FUNCTION_BLOCK CMP_OC_W4

VAR_INPUT
	BOOL_INTERLOCK : BOOL; (*INTERLOCK*)
	WORD_1: WORD;		(*WORD 1*)
	WORD_2: WORD;		(*WORD 2*)
	WORD_3: WORD;		(*WORD 3*)
	WORD_4: WORD;		(*WORD 4*)
	END_VAR


VAR_OUTPUT
	BZ_OUTPUT_BOOL : BOOL;
END_VAR


VAR
	OUT_1: BOOL;
	OUT_2: BOOL;
	OUT_3: BOOL;
	OUT_4: BOOL;
END_VAR

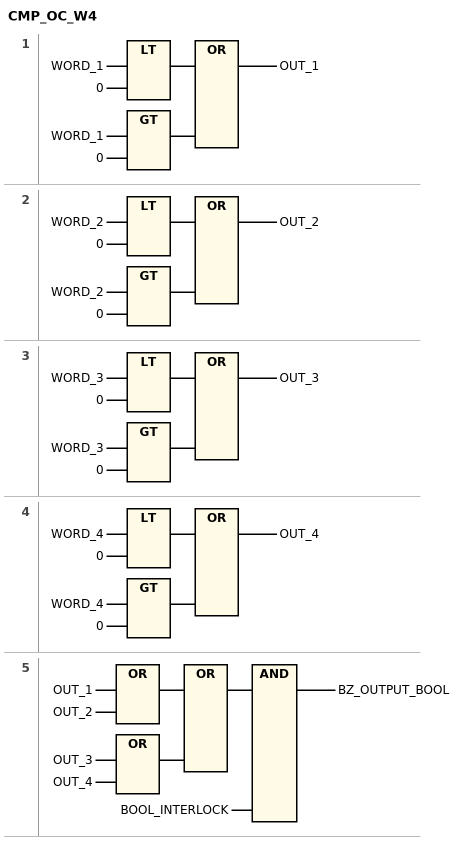
// NETWORK 1
OUT_1 := WORD_1 < 0 OR WORD_1 > 0;

// NETWORK 2
OUT_2 := WORD_2 < 0 OR WORD_2 > 0;

// NETWORK 3
OUT_3 := WORD_3 < 0 OR WORD_3 > 0;

// NETWORK 4
OUT_4 := WORD_4 < 0 OR WORD_4 > 0;

// NETWORK 5
BZ_OUTPUT_BOOL := ((OUT_1 OR OUT_2) OR (OUT_3 OR OUT_4)) AND BOOL_INTERLOCK;

END_FUNCTION_BLOCK

(* stored: Version 1.1.0.1, ProductVersion 3.1.4024.12
   POU CMP_OC_W4: Id {6aab283f-abc8-4f60-a6f2-6675e69df318}, SpecialFunc None *)
